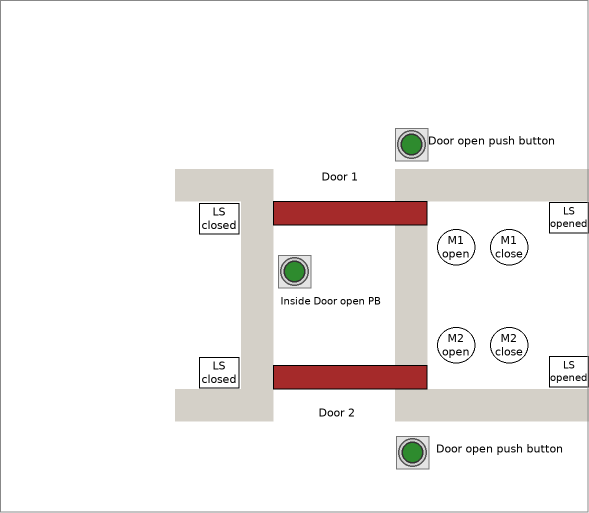
VISUALIZATION Visualization  // 589x513
    Rectangle (241,169 32x252)
    Rectangle (192,152 32x66), angle 90
    Rectangle (192,372 32x66), angle 90
    Rectangle (395,169 32x252)
    Rectangle (519,77 32x216), angle 90
    Rectangle (519,297 32x216), angle 90
    Rectangle (338,136 24x154), angle 90
        p3560616238: VisuSim.Door01Pos
    Rectangle (338,300 24x154), angle 90
        p3560616238: VisuSim.Door02Pos
    Label (309,162 62x30), "Door 1"
    Label (301,398 72x30), "Door 2"
    PushSwitch (395,126 33x37), variable: MAIN.PbOut1, behaviour: TAP, style: Switch-PushSwitch-Green
    PushSwitch (396,434 33x37), variable: MAIN.PbOut2, behaviour: TAP, style: Switch-PushSwitch-Green
    Label (421,126 141x30), "Door open push button"
    Label (429,434 141x30), "Door open push button"
    Ellipse (437,229 38x36), "M1 open", colour toggle: MAIN.MotorDoor01Open
    Ellipse (490,229 38x36), "M1 close", colour toggle: MAIN.MotorDoor01Close
    Ellipse (437,327 38x36), "M2 open", colour toggle: MAIN.MotorDoor02Open
    Ellipse (490,327 38x36), "M2 close", colour toggle: MAIN.MotorDoor02Close
    RoundedRectangle (199,203 40x31), "LS closed", colour toggle: MAIN.LsDoor1Closed
    RoundedRectangle (549,202 40x31), "LS opened", colour toggle: MAIN.LsDoor1Opened
    RoundedRectangle (199,357 40x31), "LS closed", colour toggle: MAIN.LsDoor2Closed
    RoundedRectangle (549,356 40x31), "LS opened", colour toggle: MAIN.LsDoor2Opened
    PushSwitch (278,253 33x37), variable: MAIN.PbIn1, behaviour: TAP, style: Switch-PushSwitch-Green
    Label (271,286 120x30), "Inside Door open PB"
END_VISUALIZATION

(* stored: Version 1.1.0.1, ProductVersion 3.1.4024.15
   Visu Visualization: Id {f7248a2c-f528-4b4f-bbd9-0df17197f88c} *)
